INTERFACE I_ControlBox

END_INTERFACE

(* stored: Version 1.1.0.1, ProductVersion 3.1.4024.12
   Itf I_ControlBox: Id {ce76413b-7dd4-48d6-aab8-c5d88ae23c65} *)
